FUNCTION_BLOCK XtsMoverNctTask EXTENDS XtsCore.XtsMoverTaskResult IMPLEMENTS I_XtsMoverTask, I_XtsNctMoverTask
VAR
	_Axis		: XtsCore.I_AxisRef;
	_System		: I_XtsSystem;
	_DefaultNct : XtsNctBaseUnit;
	_Nct		: I_XtsNctBaseUnit := _DefaultNct;
	_State		: UDINT;
END_VAR

PROPERTY Axis : XtsCore.I_AxisRef
GET
Axis := _Axis;
END_GET
SET
VAR
	Mover : I_XtsMover;
END_VAR
_Axis := Axis;
__QUERYINTERFACE(_Axis, Mover);
_Mover := Mover;
__QUERYINTERFACE(Mover.TracePublisher, _Logger);
END_SET
END_PROPERTY

METHOD CyclicLogic
IF _System = 0 THEN
	RETURN;
END_IF

SUPER^.CyclicLogic(); //Watchdog handling
CASE _State OF
	0:
		
		IF _Mover.MoverId = 0 THEN
			RETURN;
		END_IF

		_Nct.AssignInterface(_System.Utility.NctControllerTcIo().BaseUnitInterfaceTcIo(UDINT_TO_UINT(_Mover.MoverId)));
		_State := 1;

	1:
		_Nct.Initalize(_Nct.Status.isReadyToInitialize);
		IF _Nct.Status.isInitialized THEN
			_State := 10;
		END_IF

	10:
		IF NOT _Nct.IsInterfaceAssigned THEN
			//We shouldn't ever lose the interface mid cycle once assigned
			LogMessage.Severity	 := 4;
			LogMessage.Message	 := 'NCT Interface lost after being assigned';
			//LogMessage.MessageId := E_XtsLogMessage.MoverCommandedToHalt;
			_Logger.LogMessageInstance(LogSource, LogMessage);
			_Error := TRUE;
			_State := 0;
			RETURN;
		END_IF

		IF NOT _Nct.Status.isInitialized THEN
			_State := 1;
			RETURN;
		END_IF

		_Nct.UpdateProcessData(_Nct.Status.isOnCommunicationArea AND _Nct.Status.isReadyToProcessSyncCommands);
END_CASE
END_METHOD

METHOD Execute : I_XtsMoverTaskResult
Execute			:= THIS^;
ExecuteWatchdog := ExecuteWatchdog + 1;

//Protect against repeated calls
IF _Busy OR _CommandExecuted THEN
	RETURN;
END_IF

_Error				 := FALSE;
_ErrorID			 := 0;
_Busy				 := TRUE;
END_METHOD

//FB_Init is always available implicitly and it is used primarily for initialization.

//The return value is not evaluated. For a specific influence, you can also declare the

//methods explicitly and provide additional code there with the standard initialization

//code. You can evaluate the return value.
METHOD FB_Init : BOOL
VAR_INPUT
	bInitRetains : BOOL; // TRUE: the retain variables are initialized (reset warm / reset cold)
	bInCopyCode	 : BOOL; // TRUE: the instance will be copied to the copy code afterward (online change)
END_VAR
_TaskName			 := 'Nct Cyclic';
_TaskId				 := MoverTaskId.NCT; 
LogSource.SourceName := _TaskName;
LogSource.SourceId	 := _TaskId;
END_METHOD

PROPERTY Interrupted : BOOL
GET
VAR
	Mover : I_XtsMover;
END_VAR
Interrupted := FALSE;
END_GET
END_PROPERTY

{attribute 'monitoring' := 'call'}
PROPERTY Nct : I_XtsNctBaseUnit
GET
END_GET
SET
_Nct := Nct;
END_SET
END_PROPERTY

{attribute 'monitoring' := 'call'}
PROPERTY NctReady : BOOL
GET
NctReady := _Nct.IsInterfaceAssigned AND_THEN _Nct.Status.isInitialized;
END_GET
END_PROPERTY

METHOD Reset
IF _Error THEN
	_State := 0;
END_IF

_Error			 := FALSE;
_ErrorID		 := 0;
_Busy			 := FALSE;
ExecuteWatchdog	 := 0;
_CommandExecuted := FALSE;
END_METHOD

PROPERTY XtsSystem : I_XtsSystem
GET
XtsSystem := _System;
END_GET
SET
_System := XtsSystem;
END_SET
END_PROPERTY

END_FUNCTION_BLOCK

(* stored: Version 1.1.0.1, ProductVersion 3.1.4026.19
   POU XtsMoverNctTask: Id {c4d6f204-c5c0-4759-aac5-41330eed750b}, SpecialFunc None
   Folder Constructor: Id {f89fc7eb-cb1b-4603-b4dd-869c20756a02}
   Property Axis: Id {6e38082e-2782-407d-877b-c66258cf1236}
   Get Get: Id {a596a4fa-21e9-4ccc-bbab-6d3f378326d3}
   Set Set: Id {558d6dff-fdab-4c3e-a42b-f2d11bf57397}
   Method CyclicLogic: Id {f2a170b2-9336-437d-bac4-2559323b9c3f}
   Method Execute: Id {8998026a-5464-41fa-9a46-dbc499eba7d1}
   Method FB_Init: Id {36ffd55e-fa41-401d-91b6-a081ca3156ce}
   Property Interrupted: Id {5be10101-c763-46ba-8c84-de7f90c6b855}
   Get Get: Id {1d06db6a-b74a-4385-9668-6cf408337f9b}
   Property Nct: Id {87e666f2-f7d8-4bf2-82b7-e683a7eb82c8}
   Get Get: Id {9081d5ee-4c26-400f-b51c-d8edf2e724d8}
   Set Set: Id {29640f25-eec5-446a-a15b-8ed93c591ac2}
   Property NctReady: Id {4320834d-b216-47cd-827e-200045134ce6}
   Get Get: Id {ad43369f-4705-42ae-88d7-f8b093c950ac}
   Method Reset: Id {b6394ab1-0ee2-4242-b5c7-d79a497c5b3e}
   Property XtsSystem: Id {4f160afa-d37b-4280-b162-cd8617a56d2e}
   Get Get: Id {d9cda854-b17f-4f53-9c4b-27cc162f67d0}
   Set Set: Id {b1b77ff1-8660-4009-a8f4-68d739f7587c} *)
